// TIA Portal V19 export
DATA_BLOCK "AUTO SUBOUTPUT DB"   // DB46
{ S7_Optimized_Access := 'TRUE' }
// stored: MemoryReserve 100
   VAR
      "SYRUP MFG VESSEL BOTTOM STERROR RUN" : Bool;
      "PREMIXING VESSEL BOTTOM STERROR RUN" : Bool;
      "INLINE 1 HOMOGENIZER MOTOR1 RUN" : Bool;
      "INLINE 2 HOMOGENIZER MOTOR 2 RUN" : Bool;
      "FILTER PRESS MOTOR 1 RUN" : Bool;
      "FILTER PRESS MOTOR 2 RUN" : Bool;
      "VACCUM PUMP MOTOR-W 1 RUN" : Bool;
      "VACCUMP PUMP MOTOR-S2 RUN" : Bool;
      "VACCUMP PUMP MOTOR-W 3 RUN" : Bool;
      "VACCUMP PUMP MOTOR-S 4 RUN" : Bool;
      "SUGAR VESSEL BOTTOM STERROR RUN" : Bool;
      "BASKET FILTER MOTOR RUN" : Bool;
      "PBV-01 INGREDIENT INLET" : Bool;
      "PBV-02 CIP INLET (SPRAY BALL)" : Bool;
      "PBV-03 VENT FILTER ISOLATION" : Bool;
      "PBV-04 PW INLET" : Bool;
      "PBV-07 PREMIX TANK DRAIN VALVE" : Bool;
      "PAV-09 JACKET STEAM INLET" : Bool;
      "PAV-10 JACKET CONDENSATE DRAIN" : Bool;
      "PAV-11 JACKET BYPASS DRAIN VALVE" : Bool;
      "PAV-12 SEAL COOLING INLET" : Bool;
      "PAV-13 WATER COOLING INLET" : Bool;
      "PAV-14 WATER COOLING OUTLET" : Bool;
      "PBV-15 VACUUM INLET" : Bool;
      "PBV-16 VACUUM VENT VALVE" : Bool;
      "PFBV-17 TANK OUTLET VALVE" : Bool;
      "PBV-19 PW INLET" : Bool;
      "PBV-20 CIP INLET (SPRAY BALL)" : Bool;
      "PBV-21 VENT FILTER ISOLATION" : Bool;
      "PBV-22 INGREDIENT INLET (SUGAR INLET)" : Bool;
      "PBV-25 BOTTOM OUTLET TO DRAIN VALVE" : Bool;
      "PAV-27 JACKET STEAM INLET" : Bool;
      "PAV-28 SEAL COOLING INLET" : Bool;
      "PAV-29 JACKET CONDENSATE DRAIN" : Bool;
      "PBV-30 VACUUM INLET VALVE" : Bool;
      "PBV-31 VACUUM VENT VALVE" : Bool;
      "PFBV-32 TANK OUTLET VALVE" : Bool;
      "PBV-36 PW INLET" : Bool;
      "PBV-37 VENT FILTER ISOLATION" : Bool;
      "PBV-38 CIP INLET LINE" : Bool;
      "PBV-41 MFG TANK DRAIN VALVE" : Bool;
      "PAV-50 JACKET STEAM INLET" : Bool;
      "PAV-51 WATER COOLING OUTLET" : Bool;
      "PAV-52 WATER COOLING INLET" : Bool;
      "PAV-53 SEAL COOLING INLET" : Bool;
      "PAV-54 JACKET STEAM OUTLET VALVE" : Bool;
      "PAV-55 JACKET CONDENSATE BYPASS DRAIN" : Bool;
      "PAV-56 INLINE HOMO. SEAL COOLING INLET" : Bool;
      "PBV-57 VACUUM INLET VALVE" : Bool;
      "PFBV-59 TANK OUTLET VALVE" : Bool;
      "PBV-79 BASKET FILTER INLET" : Bool;
      "PBV-80 BOTTOM OUTLET TO BASKET FILTER" : Bool;
      "PBV-81 TANK BOTTOM OUTLET TO CIP OUTLET" : Bool;
      "PBV-82 CIP ISOLATION" : Bool;
      "PBV-83 PREMIX TRANSFER TO MFG VESSEL TRANSFER (TOP DISH)" : Bool;
      "PBV-84 FROM TANK OUTLET TO CIP OUTLET" : Bool;
      "PBV-85 SORBITOL INLET LINE" : Bool;
      "PBV-86 GLUCOSE INLET LINE" : Bool;
      "PBV-87 BASKET FILTER TO PREMIX VESSEL LINE" : Bool;
      "PBV-88 BASKET FILTER TRANSFER LINE" : Bool;
      "PBV-89 BASKET FILTER TO MFG INLET TRANSFER LINE" : Bool;
      "PBV-90 PREMIX TO MFG TRANSFER LINE" : Bool;
      "PBV-91 PREMIX TO MFG TRANSFER LINE" : Bool;
      "PBV-92 PREMIX TO STORAGE – 4 TRANSFER LINE" : Bool;
      "PBV-93 TANK OUTLET TO INLINE HOMOGENIZER LINE" : Bool;
      "PBV-94 INLINE HOMOGENIZER INLET LINE" : Bool;
      "PBV-95 TANK OUTLET TO FILTER PRESS LINE" : Bool;
      "PBV-96 INLINE HOMOGENIZER RECIRCULATION LINE" : Bool;
      "PBV-97 FILTER PRESS OUTLET" : Bool;
      "PBV-98 INLINE HOMOGENIZER TO FILTER PRESS OUTLET LINE" : Bool;
      "PAV-99 INLINE HOMOGENIZER SEAL COOLING" : Bool;
      "PBV-100 FILTER PRESS INLET" : Bool;
      "PBV-101 SUGAR MELTING TO MFG TRANSFER (TOP DISH)" : Bool;
      "PBV-102 PREMIX TO MFG TRANSFER (TOP DISH)" : Bool;
      "PBV-103 CIP INLET (SPRAY BALL)" : Bool;
      "PBV-104 MFG VESSEL TRANSFER LINE" : Bool;
      "PBV-105 INGREDIENT INLET" : Bool;
      "PBV-106 SORBITOL INLET" : Bool;
      "PBV-107 GLUCOSE INLET" : Bool;
      "PBV-108 INLINE HOMOGENIZER TO FILTER PRESS INLET LINE" : Bool;
      "PBV-109 HOMO. RECIRCULATION INLET" : Bool;
      "PBV-110 INLINE HOMOGENIZER TO INLET LINE" : Bool;
      "PBV-111 FILTER PRESS OUTLER VALVE" : Bool;
      "PBV-112 FILTER PRESS TO TRANSFER LINE" : Bool;
      "PAV-113 TANK OUTLET TO CIP DRAIN LINE" : Bool;
      "PBV-114 TANK OUTLET TO INLINE HOMOGENIZER LINE" : Bool;
      "PBV-115 MFG TO STORAGE – 1 TRANSFER LINE" : Bool;
      "PBV-116 MFG TO STORAGE – 2 TRANSFER LINE" : Bool;
      "PBV-117 MFG TO STORAGE – 3 TRANSFER LINE" : Bool;
      "PBV-118 FILTER PRESS INLET" : Bool;
      "PBV-119 SEAL COOLING FOR STORAGE VESSEL - 4" : Bool;
      "PBV-120 SEAL COOLING FOR STORAGE VESSEL - 3" : Bool;
      "PBV-121 SEAL COOLING FOR STORAGE VESSEL - 2" : Bool;
      "PBV-122 SEAL COOLING FOR STORAGE VESSEL - 1" : Bool;
      "PBV-123 VESSEL TOP DISH" : Bool;
      "PBV-124 VESSEL INLET LINE" : Bool;
      "PBV-149" : Bool;
      "PBV-150" : Bool;
      "PBV-151" : Bool;
      "PBV-152" : Bool;
      "PBV-153" : Bool;
      "PBV-155" : Bool;
      "PBV-156" : Bool;
   END_VAR
BEGIN
END_DATA_BLOCK
